FUNCTION_BLOCK PUBLIC TOD_TO_TestSuite EXTENDS TcUnit.FB_TestSuite
VAR
END_VAR

Check_TOD_TO_BOOL_Max();
Check_TOD_TO_BOOL_Min();
Check_TOD_TO_BYTE_Max();
Check_TOD_TO_BYTE_Min();
Check_TOD_TO_BYTE_TooHigh();
Check_TOD_TO_WORD_Max();
Check_TOD_TO_WORD_Min();
Check_TOD_TO_WORD_TooHigh();
Check_TOD_TO_DWORD_Max();
Check_TOD_TO_DWORD_Min();
Check_TOD_TO_LWORD_Max();
Check_TOD_TO_LWORD_Min();
Check_TOD_TO_SINT_Max();
Check_TOD_TO_SINT_Min();
Check_TOD_TO_SINT_TooHigh();
Check_TOD_TO_INT_Max();
Check_TOD_TO_INT_Min();
Check_TOD_TO_INT_TooHigh();
Check_TOD_TO_DINT_Max();
Check_TOD_TO_DINT_Min();
Check_TOD_TO_LINT_Max();
Check_TOD_TO_LINT_Min();
Check_TOD_TO_USINT_Max();
Check_TOD_TO_USINT_Min();
Check_TOD_TO_USINT_TooHigh();
Check_TOD_TO_UINT_Max();
Check_TOD_TO_UINT_Min();
Check_TOD_TO_UINT_TooHigh();
Check_TOD_TO_UDINT_Max();
Check_TOD_TO_UDINT_Min();
Check_TOD_TO_ULINT_Max();
Check_TOD_TO_ULINT_Min();
Check_TOD_TO_REAL_Max();
Check_TOD_TO_REAL_Min();
Check_TOD_TO_LREAL_Max();
Check_TOD_TO_LREAL_Min();
Check_TOD_TO_TIME_Max();
Check_TOD_TO_TIME_Min();
Check_TOD_TO_TOD_Max();
Check_TOD_TO_TOD_Min();
Check_TOD_TO_DATE_Max();
Check_TOD_TO_DATE_Min();
Check_TOD_TO_DT_Max();
Check_TOD_TO_DT_Min();
Check_TOD_TO_STRING_Max();
Check_TOD_TO_STRING_Min();

METHOD PUBLIC Check_TOD_TO_BOOL_Min
VAR
	value : TOD := DatatypeLimits.TOD_MIN_VALUE;
	actual : BOOL;
	converted : BOOL;
	equal : BOOL;
END_VAR
TEST('Check_TOD_TO_BOOL_Min');

// @TEST-RUN
converted := TryConvert_TOD_TO_Destination(value, actual);
equal := actual = TOD_TO_BOOL(value);

// @TEST-ASSERT
AssertTrue(Condition := equal, Message := 'Did not convert TOD to BOOL correctly');
AssertTrue(Condition := converted, Message := 'Did not report TOD to BOOL conversion was successful');

TEST_FINISHED();
END_METHOD

METHOD PUBLIC Check_TOD_TO_BOOL_Max
VAR
	value : TOD := DatatypeLimits.TOD_MAX_VALUE;
	actual : BOOL;
	converted : BOOL;
	equal : BOOL;
END_VAR
TEST('Check_TOD_TO_BOOL_Max');

// @TEST-RUN
converted := TryConvert_TOD_TO_Destination(value, actual);
equal := actual = TOD_TO_BOOL(value);

// @TEST-ASSERT
AssertTrue(Condition := equal, Message := 'Did not convert TOD to BOOL correctly');
AssertTrue(Condition := converted, Message := 'Did not report TOD to BOOL conversion was successful');

TEST_FINISHED();
END_METHOD

METHOD PUBLIC Check_TOD_TO_BYTE_Min
VAR
	value : TOD := DatatypeLimits.TOD_MIN_VALUE;
	actual : BYTE;
	converted : BOOL;
	equal : BOOL;
END_VAR
TEST('Check_TOD_TO_BYTE_Min');

// @TEST-RUN
converted := TryConvert_TOD_TO_Destination(value, actual);
equal := actual = TOD_TO_BYTE(value);

// @TEST-ASSERT
AssertTrue(Condition := equal, Message := 'Did not convert TOD to BYTE correctly');
AssertTrue(Condition := converted, Message := 'Did not report TOD to BYTE conversion was successful');

TEST_FINISHED();
END_METHOD

METHOD PUBLIC Check_TOD_TO_BYTE_TooHigh
VAR
	value : TOD := DatatypeLimits.TOD_MAX_VALUE;
	actual : BYTE;
	converted : BOOL;
END_VAR
TEST('Check_TOD_TO_BYTE_TooHigh');

// @TEST-RUN
converted := TryConvert_TOD_TO_Destination(value, actual);

// @TEST-ASSERT
AssertFalse(Condition := converted, Message := 'Did not report TOD to BYTE conversion was prevented');

TEST_FINISHED();
END_METHOD

METHOD PUBLIC Check_TOD_TO_BYTE_Max
VAR
	value : TOD := DatatypeLimits.MAX_VALUE_OF_TOD_WHICH_CAN_BE_HELD_IN_A_BYTE;
	actual : BYTE;
	converted : BOOL;
	equal : BOOL;
END_VAR
TEST('Check_TOD_TO_BYTE_Max');

// @TEST-RUN
converted := TryConvert_TOD_TO_Destination(value, actual);
equal := actual = TOD_TO_BYTE(value);

// @TEST-ASSERT
AssertTrue(Condition := equal, Message := 'Did not convert TOD to BYTE correctly');
AssertTrue(Condition := converted, Message := 'Did not report TOD to BYTE conversion was successful');

TEST_FINISHED();
END_METHOD

METHOD PUBLIC Check_TOD_TO_DATE_Min
VAR
	value : TOD := DatatypeLimits.TOD_MIN_VALUE;
	actual : DATE;
	converted : BOOL;
	equal : BOOL;
END_VAR
TEST('Check_TOD_TO_DATE_Min');

// @TEST-RUN
converted := TryConvert_TOD_TO_Destination(value, actual);
equal := actual = TOD_TO_DATE(value);

// @TEST-ASSERT
AssertTrue(Condition := equal, Message := 'Did not convert TOD to DATE correctly');
AssertTrue(Condition := converted, Message := 'Did not report TOD to DATE conversion was successful');

TEST_FINISHED();
END_METHOD

METHOD PUBLIC Check_TOD_TO_DATE_Max
VAR
	value : TOD := DatatypeLimits.TOD_MAX_VALUE;
	actual : DATE;
	converted : BOOL;
	equal : BOOL;
END_VAR
TEST('Check_TOD_TO_DATE_Max');

// @TEST-RUN
converted := TryConvert_TOD_TO_Destination(value, actual);
equal := actual = TOD_TO_DATE(value);

// @TEST-ASSERT
AssertTrue(Condition := equal, Message := 'Did not convert TOD to DATE correctly');
AssertTrue(Condition := converted, Message := 'Did not report TOD to DATE conversion was successful');

TEST_FINISHED();
END_METHOD

METHOD PUBLIC Check_TOD_TO_DINT_Min
VAR
	value : TOD := DatatypeLimits.TOD_MIN_VALUE;
	actual : DINT;
	converted : BOOL;
	equal : BOOL;
END_VAR
TEST('Check_TOD_TO_DINT_Min');

// @TEST-RUN
converted := TryConvert_TOD_TO_Destination(value, actual);
equal := actual = TOD_TO_DINT(value);

// @TEST-ASSERT
AssertTrue(Condition := equal, Message := 'Did not convert TOD to DINT correctly');
AssertTrue(Condition := converted, Message := 'Did not report TOD to DINT conversion was successful');

TEST_FINISHED();
END_METHOD

METHOD PUBLIC Check_TOD_TO_DINT_Max
VAR
	value : TOD := DatatypeLimits.TOD_MAX_VALUE;
	actual : DINT;
	converted : BOOL;
	equal : BOOL;
END_VAR
TEST('Check_TOD_TO_DINT_Max');

// @TEST-RUN
converted := TryConvert_TOD_TO_Destination(value, actual);
equal := actual = TOD_TO_DINT(value);

// @TEST-ASSERT
AssertTrue(Condition := equal, Message := 'Did not convert TOD to DINT correctly');
AssertTrue(Condition := converted, Message := 'Did not report TOD to DINT conversion was successful');

TEST_FINISHED();
END_METHOD

METHOD PUBLIC Check_TOD_TO_DT_Min
VAR
	value : TOD := DatatypeLimits.TOD_MIN_VALUE;
	actual : DT;
	converted : BOOL;
	equal : BOOL;
END_VAR
TEST('Check_TOD_TO_DT_Min');

// @TEST-RUN
converted := TryConvert_TOD_TO_Destination(value, actual);
equal := actual = TOD_TO_DT(value);

// @TEST-ASSERT
AssertTrue(Condition := equal, Message := 'Did not convert TOD to DT correctly');
AssertTrue(Condition := converted, Message := 'Did not report TOD to DT conversion was successful');

TEST_FINISHED();
END_METHOD

METHOD PUBLIC Check_TOD_TO_DT_Max
VAR
	value : TOD := DatatypeLimits.TOD_MAX_VALUE;
	actual : DT;
	converted : BOOL;
	equal : BOOL;
END_VAR
TEST('Check_TOD_TO_DT_Max');

// @TEST-RUN
converted := TryConvert_TOD_TO_Destination(value, actual);
equal := actual = TOD_TO_DT(value);

// @TEST-ASSERT
AssertTrue(Condition := equal, Message := 'Did not convert TOD to DT correctly');
AssertTrue(Condition := converted, Message := 'Did not report TOD to DT conversion was successful');

TEST_FINISHED();
END_METHOD

METHOD PUBLIC Check_TOD_TO_DWORD_Min
VAR
	value : TOD := DatatypeLimits.TOD_MIN_VALUE;
	actual : DWORD;
	converted : BOOL;
	equal : BOOL;
END_VAR
TEST('Check_TOD_TO_DWORD_Min');

// @TEST-RUN
converted := TryConvert_TOD_TO_Destination(value, actual);
equal := actual = TOD_TO_DWORD(value);

// @TEST-ASSERT
AssertTrue(Condition := equal, Message := 'Did not convert TOD to DWORD correctly');
AssertTrue(Condition := converted, Message := 'Did not report TOD to DWORD conversion was successful');

TEST_FINISHED();
END_METHOD

METHOD PUBLIC Check_TOD_TO_DWORD_Max
VAR
	value : TOD := DatatypeLimits.TOD_MAX_VALUE;
	actual : DWORD;
	converted : BOOL;
	equal : BOOL;
END_VAR
TEST('Check_TOD_TO_DWORD_Max');

// @TEST-RUN
converted := TryConvert_TOD_TO_Destination(value, actual);
equal := actual = TOD_TO_DWORD(value);

// @TEST-ASSERT
AssertTrue(Condition := equal, Message := 'Did not convert TOD to DWORD correctly');
AssertTrue(Condition := converted, Message := 'Did not report TOD to DWORD conversion was successful');

TEST_FINISHED();
END_METHOD

METHOD PUBLIC Check_TOD_TO_INT_Min
VAR
	value : TOD := DatatypeLimits.TOD_MIN_VALUE;
	actual : INT;
	converted : BOOL;
	equal : BOOL;
END_VAR
TEST('Check_TOD_TO_INT_Min');

// @TEST-RUN
converted := TryConvert_TOD_TO_Destination(value, actual);
equal := actual = TOD_TO_INT(value);

// @TEST-ASSERT
AssertTrue(Condition := equal, Message := 'Did not convert TOD to INT correctly');
AssertTrue(Condition := converted, Message := 'Did not report TOD to INT conversion was successful');

TEST_FINISHED();
END_METHOD

METHOD PUBLIC Check_TOD_TO_INT_TooHigh
VAR
	value : TOD := DatatypeLimits.TOD_MAX_VALUE;
	actual : INT;
	converted : BOOL;
END_VAR
TEST('Check_TOD_TO_INT_TooHigh');

// @TEST-RUN
converted := TryConvert_TOD_TO_Destination(value, actual);

// @TEST-ASSERT
AssertFalse(Condition := converted, Message := 'Did not report TOD to INT conversion was prevented');

TEST_FINISHED();
END_METHOD

METHOD PUBLIC Check_TOD_TO_INT_Max
VAR
	value : TOD := DatatypeLimits.MAX_VALUE_OF_TOD_WHICH_CAN_BE_HELD_IN_A_INT;
	actual : INT;
	converted : BOOL;
	equal : BOOL;
END_VAR
TEST('Check_TOD_TO_INT_Max');

// @TEST-RUN
converted := TryConvert_TOD_TO_Destination(value, actual);
equal := actual = TOD_TO_INT(value);

// @TEST-ASSERT
AssertTrue(Condition := equal, Message := 'Did not convert TOD to INT correctly');
AssertTrue(Condition := converted, Message := 'Did not report TOD to INT conversion was successful');

TEST_FINISHED();
END_METHOD

METHOD PUBLIC Check_TOD_TO_LINT_Min
VAR
	value : TOD := DatatypeLimits.TOD_MIN_VALUE;
	actual : LINT;
	converted : BOOL;
	equal : BOOL;
END_VAR
TEST('Check_TOD_TO_LINT_Min');

// @TEST-RUN
converted := TryConvert_TOD_TO_Destination(value, actual);
equal := actual = TOD_TO_LINT(value);

// @TEST-ASSERT
AssertTrue(Condition := equal, Message := 'Did not convert TOD to LINT correctly');
AssertTrue(Condition := converted, Message := 'Did not report TOD to LINT conversion was successful');

TEST_FINISHED();
END_METHOD

METHOD PUBLIC Check_TOD_TO_LINT_Max
VAR
	value : TOD := DatatypeLimits.TOD_MAX_VALUE;
	actual : LINT;
	converted : BOOL;
	equal : BOOL;
END_VAR
TEST('Check_TOD_TO_LINT_Max');

// @TEST-RUN
converted := TryConvert_TOD_TO_Destination(value, actual);
equal := actual = TOD_TO_LINT(value);

// @TEST-ASSERT
AssertTrue(Condition := equal, Message := 'Did not convert TOD to LINT correctly');
AssertTrue(Condition := converted, Message := 'Did not report TOD to LINT conversion was successful');

TEST_FINISHED();
END_METHOD

METHOD PUBLIC Check_TOD_TO_LREAL_Min
VAR
	value : TOD := DatatypeLimits.TOD_MIN_VALUE;
	actual : LREAL;
	converted : BOOL;
	equal : BOOL;
END_VAR
TEST('Check_TOD_TO_LREAL_Min');

// @TEST-RUN
converted := TryConvert_TOD_TO_Destination(value, actual);
equal := actual = TOD_TO_LREAL(value);

// @TEST-ASSERT
AssertTrue(Condition := equal, Message := 'Did not convert TOD to LREAL correctly');
AssertTrue(Condition := converted, Message := 'Did not report TOD to LREAL conversion was successful');

TEST_FINISHED();
END_METHOD

METHOD PUBLIC Check_TOD_TO_LREAL_Max
VAR
	value : TOD := DatatypeLimits.TOD_MAX_VALUE;
	actual : LREAL;
	converted : BOOL;
	equal : BOOL;
END_VAR
TEST('Check_TOD_TO_LREAL_Max');

// @TEST-RUN
converted := TryConvert_TOD_TO_Destination(value, actual);
equal := actual = TOD_TO_LREAL(value);

// @TEST-ASSERT
AssertTrue(Condition := equal, Message := 'Did not convert TOD to LREAL correctly');
AssertTrue(Condition := converted, Message := 'Did not report TOD to LREAL conversion was successful');

TEST_FINISHED();
END_METHOD

METHOD PUBLIC Check_TOD_TO_LWORD_Min
VAR
	value : TOD := DatatypeLimits.TOD_MIN_VALUE;
	actual : LWORD;
	converted : BOOL;
	equal : BOOL;
END_VAR
TEST('Check_TOD_TO_LWORD_Min');

// @TEST-RUN
converted := TryConvert_TOD_TO_Destination(value, actual);
equal := actual = TOD_TO_LWORD(value);

// @TEST-ASSERT
AssertTrue(Condition := equal, Message := 'Did not convert TOD to LWORD correctly');
AssertTrue(Condition := converted, Message := 'Did not report TOD to LWORD conversion was successful');

TEST_FINISHED();
END_METHOD

METHOD PUBLIC Check_TOD_TO_LWORD_Max
VAR
	value : TOD := DatatypeLimits.TOD_MAX_VALUE;
	actual : LWORD;
	converted : BOOL;
	equal : BOOL;
END_VAR
TEST('Check_TOD_TO_LWORD_Max');

// @TEST-RUN
converted := TryConvert_TOD_TO_Destination(value, actual);
equal := actual = TOD_TO_LWORD(value);

// @TEST-ASSERT
AssertTrue(Condition := equal, Message := 'Did not convert TOD to LWORD correctly');
AssertTrue(Condition := converted, Message := 'Did not report TOD to LWORD conversion was successful');

TEST_FINISHED();
END_METHOD

METHOD PUBLIC Check_TOD_TO_REAL_Min
VAR
	value : TOD := DatatypeLimits.TOD_MIN_VALUE;
	actual : REAL;
	converted : BOOL;
	equal : BOOL;
END_VAR
TEST('Check_TOD_TO_REAL_Min');

// @TEST-RUN
converted := TryConvert_TOD_TO_Destination(value, actual);
equal := actual = TOD_TO_REAL(value);

// @TEST-ASSERT
AssertTrue(Condition := equal, Message := 'Did not convert TOD to REAL correctly');
AssertTrue(Condition := converted, Message := 'Did not report TOD to REAL conversion was successful');

TEST_FINISHED();
END_METHOD

METHOD PUBLIC Check_TOD_TO_REAL_Max
VAR
	value : TOD := DatatypeLimits.TOD_MAX_VALUE;
	actual : REAL;
	converted : BOOL;
	equal : BOOL;
END_VAR
TEST('Check_TOD_TO_REAL_Max');

// @TEST-RUN
converted := TryConvert_TOD_TO_Destination(value, actual);
equal := actual = TOD_TO_REAL(value);

// @TEST-ASSERT
AssertTrue(Condition := equal, Message := 'Did not convert TOD to REAL correctly');
AssertTrue(Condition := converted, Message := 'Did not report TOD to REAL conversion was successful');

TEST_FINISHED();
END_METHOD

METHOD PUBLIC Check_TOD_TO_SINT_Min
VAR
	value : TOD := DatatypeLimits.TOD_MIN_VALUE;
	actual : SINT;
	converted : BOOL;
	equal : BOOL;
END_VAR
TEST('Check_TOD_TO_SINT_Min');

// @TEST-RUN
converted := TryConvert_TOD_TO_Destination(value, actual);
equal := actual = TOD_TO_SINT(value);

// @TEST-ASSERT
AssertTrue(Condition := equal, Message := 'Did not convert TOD to SINT correctly');
AssertTrue(Condition := converted, Message := 'Did not report TOD to SINT conversion was successful');

TEST_FINISHED();
END_METHOD

METHOD PUBLIC Check_TOD_TO_SINT_TooHigh
VAR
	value : TOD := DatatypeLimits.TOD_MAX_VALUE;
	actual : SINT;
	converted : BOOL;
END_VAR
TEST('Check_TOD_TO_SINT_TooHigh');

// @TEST-RUN
converted := TryConvert_TOD_TO_Destination(value, actual);

// @TEST-ASSERT
AssertFalse(Condition := converted, Message := 'Did not report TOD to SINT conversion was prevented');

TEST_FINISHED();
END_METHOD

METHOD PUBLIC Check_TOD_TO_SINT_Max
VAR
	value : TOD := DatatypeLimits.MAX_VALUE_OF_TOD_WHICH_CAN_BE_HELD_IN_A_SINT;
	actual : SINT;
	converted : BOOL;
	equal : BOOL;
END_VAR
TEST('Check_TOD_TO_SINT_Max');

// @TEST-RUN
converted := TryConvert_TOD_TO_Destination(value, actual);
equal := actual = TOD_TO_SINT(value);

// @TEST-ASSERT
AssertTrue(Condition := equal, Message := 'Did not convert TOD to SINT correctly');
AssertTrue(Condition := converted, Message := 'Did not report TOD to SINT conversion was successful');

TEST_FINISHED();
END_METHOD

METHOD PUBLIC Check_TOD_TO_STRING_Min
VAR
	value : TOD := DatatypeLimits.TOD_MIN_VALUE;
	actual : STRING;
	converted : BOOL;
	equal : BOOL;
END_VAR
TEST('Check_TOD_TO_STRING_Min');

// @TEST-RUN
converted := TryConvert_TOD_TO_Destination(value, actual);
equal := actual = TOD_TO_STRING(value);

// @TEST-ASSERT
AssertTrue(Condition := equal, Message := 'Did not convert TOD to STRING correctly');
AssertTrue(Condition := converted, Message := 'Did not report TOD to STRING conversion was successful');

TEST_FINISHED();
END_METHOD

METHOD PUBLIC Check_TOD_TO_STRING_Max
VAR
	value : TOD := DatatypeLimits.TOD_MAX_VALUE;
	actual : STRING;
	converted : BOOL;
	equal : BOOL;
END_VAR
TEST('Check_TOD_TO_STRING_Max');

// @TEST-RUN
converted := TryConvert_TOD_TO_Destination(value, actual);
equal := actual = TOD_TO_STRING(value);

// @TEST-ASSERT
AssertTrue(Condition := equal, Message := 'Did not convert TOD to STRING correctly');
AssertTrue(Condition := converted, Message := 'Did not report TOD to STRING conversion was successful');

TEST_FINISHED();
END_METHOD

METHOD PUBLIC Check_TOD_TO_TIME_Min
VAR
	value : TOD := DatatypeLimits.TOD_MIN_VALUE;
	actual : TIME;
	converted : BOOL;
	equal : BOOL;
END_VAR
TEST('Check_TOD_TO_TIME_Min');

// @TEST-RUN
converted := TryConvert_TOD_TO_Destination(value, actual);
equal := actual = TOD_TO_TIME(value);

// @TEST-ASSERT
AssertTrue(Condition := equal, Message := 'Did not convert TOD to TIME correctly');
AssertTrue(Condition := converted, Message := 'Did not report TOD to TIME conversion was successful');

TEST_FINISHED();
END_METHOD

METHOD PUBLIC Check_TOD_TO_TIME_Max
VAR
	value : TOD := DatatypeLimits.TOD_MAX_VALUE;
	actual : TIME;
	converted : BOOL;
	equal : BOOL;
END_VAR
TEST('Check_TOD_TO_TIME_Max');

// @TEST-RUN
converted := TryConvert_TOD_TO_Destination(value, actual);
equal := actual = TOD_TO_TIME(value);

// @TEST-ASSERT
AssertTrue(Condition := equal, Message := 'Did not convert TOD to TIME correctly');
AssertTrue(Condition := converted, Message := 'Did not report TOD to TIME conversion was successful');

TEST_FINISHED();
END_METHOD

METHOD PUBLIC Check_TOD_TO_TOD_Min
VAR
	value : TOD := DatatypeLimits.TOD_MIN_VALUE;
	actual : TOD;
	converted : BOOL;
	equal : BOOL;
END_VAR
TEST('Check_TOD_TO_TOD_Min');

// @TEST-RUN
converted := TryConvert_TOD_TO_Destination(value, actual);
equal := actual = value;

// @TEST-ASSERT
AssertTrue(Condition := equal, Message := 'Did not convert TOD to TOD correctly');
AssertTrue(Condition := converted, Message := 'Did not report TOD to TOD conversion was successful');

TEST_FINISHED();
END_METHOD

METHOD PUBLIC Check_TOD_TO_TOD_Max
VAR
	value : TOD := DatatypeLimits.TOD_MAX_VALUE;
	actual : TOD;
	converted : BOOL;
	equal : BOOL;
END_VAR
TEST('Check_TOD_TO_TOD_Max');

// @TEST-RUN
converted := TryConvert_TOD_TO_Destination(value, actual);
equal := actual = value;

// @TEST-ASSERT
AssertTrue(Condition := equal, Message := 'Did not convert TOD to TOD correctly');
AssertTrue(Condition := converted, Message := 'Did not report TOD to TOD conversion was successful');

TEST_FINISHED();
END_METHOD

METHOD PUBLIC Check_TOD_TO_UDINT_Min
VAR
	value : TOD := DatatypeLimits.TOD_MIN_VALUE;
	actual : UDINT;
	converted : BOOL;
	equal : BOOL;
END_VAR
TEST('Check_TOD_TO_UDINT_Min');

// @TEST-RUN
converted := TryConvert_TOD_TO_Destination(value, actual);
equal := actual = TOD_TO_UDINT(value);

// @TEST-ASSERT
AssertTrue(Condition := equal, Message := 'Did not convert TOD to UDINT correctly');
AssertTrue(Condition := converted, Message := 'Did not report TOD to UDINT conversion was successful');

TEST_FINISHED();
END_METHOD

METHOD PUBLIC Check_TOD_TO_UDINT_Max
VAR
	value : TOD := DatatypeLimits.TOD_MAX_VALUE;
	actual : UDINT;
	converted : BOOL;
	equal : BOOL;
END_VAR
TEST('Check_TOD_TO_UDINT_Max');

// @TEST-RUN
converted := TryConvert_TOD_TO_Destination(value, actual);
equal := actual = TOD_TO_UDINT(value);

// @TEST-ASSERT
AssertTrue(Condition := equal, Message := 'Did not convert TOD to UDINT correctly');
AssertTrue(Condition := converted, Message := 'Did not report TOD to UDINT conversion was successful');

TEST_FINISHED();
END_METHOD

METHOD PUBLIC Check_TOD_TO_UINT_Min
VAR
	value : TOD := DatatypeLimits.TOD_MIN_VALUE;
	actual : UINT;
	converted : BOOL;
	equal : BOOL;
END_VAR
TEST('Check_TOD_TO_UINT_Min');

// @TEST-RUN
converted := TryConvert_TOD_TO_Destination(value, actual);
equal := actual = TOD_TO_UINT(value);

// @TEST-ASSERT
AssertTrue(Condition := equal, Message := 'Did not convert TOD to UINT correctly');
AssertTrue(Condition := converted, Message := 'Did not report TOD to UINT conversion was successful');

TEST_FINISHED();
END_METHOD

METHOD PUBLIC Check_TOD_TO_UINT_TooHigh
VAR
	value : TOD := DatatypeLimits.TOD_MAX_VALUE;
	actual : UINT;
	converted : BOOL;
END_VAR
TEST('Check_TOD_TO_UINT_TooHigh');

// @TEST-RUN
converted := TryConvert_TOD_TO_Destination(value, actual);

// @TEST-ASSERT
AssertFalse(Condition := converted, Message := 'Did not report TOD to UINT conversion was prevented');

TEST_FINISHED();
END_METHOD

METHOD PUBLIC Check_TOD_TO_UINT_Max
VAR
	value : TOD := DatatypeLimits.MAX_VALUE_OF_TOD_WHICH_CAN_BE_HELD_IN_A_UINT;
	actual : UINT;
	converted : BOOL;
	equal : BOOL;
END_VAR
TEST('Check_TOD_TO_UINT_Max');

// @TEST-RUN
converted := TryConvert_TOD_TO_Destination(value, actual);
equal := actual = TOD_TO_UINT(value);

// @TEST-ASSERT
AssertTrue(Condition := equal, Message := 'Did not convert TOD to UINT correctly');
AssertTrue(Condition := converted, Message := 'Did not report TOD to UINT conversion was successful');

TEST_FINISHED();
END_METHOD

METHOD PUBLIC Check_TOD_TO_ULINT_Min
VAR
	value : TOD := DatatypeLimits.TOD_MIN_VALUE;
	actual : ULINT;
	converted : BOOL;
	equal : BOOL;
END_VAR
TEST('Check_TOD_TO_ULINT_Min');

// @TEST-RUN
converted := TryConvert_TOD_TO_Destination(value, actual);
equal := actual = TOD_TO_ULINT(value);

// @TEST-ASSERT
AssertTrue(Condition := equal, Message := 'Did not convert TOD to ULINT correctly');
AssertTrue(Condition := converted, Message := 'Did not report TOD to ULINT conversion was successful');

TEST_FINISHED();
END_METHOD

METHOD PUBLIC Check_TOD_TO_ULINT_Max
VAR
	value : TOD := DatatypeLimits.TOD_MAX_VALUE;
	actual : ULINT;
	converted : BOOL;
	equal : BOOL;
END_VAR
TEST('Check_TOD_TO_ULINT_Max');

// @TEST-RUN
converted := TryConvert_TOD_TO_Destination(value, actual);
equal := actual = TOD_TO_ULINT(value);

// @TEST-ASSERT
AssertTrue(Condition := equal, Message := 'Did not convert TOD to ULINT correctly');
AssertTrue(Condition := converted, Message := 'Did not report TOD to ULINT conversion was successful');

TEST_FINISHED();
END_METHOD

METHOD PUBLIC Check_TOD_TO_USINT_Min
VAR
	value : TOD := DatatypeLimits.TOD_MIN_VALUE;
	actual : USINT;
	converted : BOOL;
	equal : BOOL;
END_VAR
TEST('Check_TOD_TO_USINT_Min');

// @TEST-RUN
converted := TryConvert_TOD_TO_Destination(value, actual);
equal := actual = TOD_TO_USINT(value);

// @TEST-ASSERT
AssertTrue(Condition := equal, Message := 'Did not convert TOD to USINT correctly');
AssertTrue(Condition := converted, Message := 'Did not report TOD to USINT conversion was successful');

TEST_FINISHED();
END_METHOD

METHOD PUBLIC Check_TOD_TO_USINT_TooHigh
VAR
	value : TOD := DatatypeLimits.TOD_MAX_VALUE;
	actual : USINT;
	converted : BOOL;
END_VAR
TEST('Check_TOD_TO_USINT_TooHigh');

// @TEST-RUN
converted := TryConvert_TOD_TO_Destination(value, actual);

// @TEST-ASSERT
AssertFalse(Condition := converted, Message := 'Did not report TOD to USINT conversion was prevented');

TEST_FINISHED();
END_METHOD

METHOD PUBLIC Check_TOD_TO_USINT_Max
VAR
	value : TOD := DatatypeLimits.MAX_VALUE_OF_TOD_WHICH_CAN_BE_HELD_IN_A_USINT;
	actual : USINT;
	converted : BOOL;
	equal : BOOL;
END_VAR
TEST('Check_TOD_TO_USINT_Max');

// @TEST-RUN
converted := TryConvert_TOD_TO_Destination(value, actual);
equal := actual = TOD_TO_USINT(value);

// @TEST-ASSERT
AssertTrue(Condition := equal, Message := 'Did not convert TOD to USINT correctly');
AssertTrue(Condition := converted, Message := 'Did not report TOD to USINT conversion was successful');

TEST_FINISHED();
END_METHOD

METHOD PUBLIC Check_TOD_TO_WORD_Min
VAR
	value : TOD := DatatypeLimits.TOD_MIN_VALUE;
	actual : WORD;
	converted : BOOL;
	equal : BOOL;
END_VAR
TEST('Check_TOD_TO_WORD_Min');

// @TEST-RUN
converted := TryConvert_TOD_TO_Destination(value, actual);
equal := actual = TOD_TO_WORD(value);

// @TEST-ASSERT
AssertTrue(Condition := equal, Message := 'Did not convert TOD to WORD correctly');
AssertTrue(Condition := converted, Message := 'Did not report TOD to WORD conversion was successful');

TEST_FINISHED();
END_METHOD

METHOD PUBLIC Check_TOD_TO_WORD_TooHigh
VAR
	value : TOD := DatatypeLimits.TOD_MAX_VALUE;
	actual : WORD;
	converted : BOOL;
END_VAR
TEST('Check_TOD_TO_WORD_TooHigh');

// @TEST-RUN
converted := TryConvert_TOD_TO_Destination(value, actual);

// @TEST-ASSERT
AssertFalse(Condition := converted, Message := 'Did not report TOD to WORD conversion was prevented');

TEST_FINISHED();
END_METHOD

METHOD PUBLIC Check_TOD_TO_WORD_Max
VAR
	value : TOD := DatatypeLimits.MAX_VALUE_OF_TOD_WHICH_CAN_BE_HELD_IN_A_WORD;
	actual : WORD;
	converted : BOOL;
	equal : BOOL;
END_VAR
TEST('Check_TOD_TO_WORD_Max');

// @TEST-RUN
converted := TryConvert_TOD_TO_Destination(value, actual);
equal := actual = TOD_TO_WORD(value);

// @TEST-ASSERT
AssertTrue(Condition := equal, Message := 'Did not convert TOD to WORD correctly');
AssertTrue(Condition := converted, Message := 'Did not report TOD to WORD conversion was successful');

TEST_FINISHED();
END_METHOD

END_FUNCTION_BLOCK

(* stored: Version 1.1.0.1, ProductVersion 3.1.4024.12
   POU TOD_TO_TestSuite: Id {268fba33-c979-45d2-9197-3ae649925bde}, SpecialFunc None
   Method Check_TOD_TO_BOOL_Min: Id {aa227d84-f942-4487-8b06-d71c2117467e}
   Method Check_TOD_TO_BOOL_Max: Id {ccc2f7bd-7b2e-43f1-8674-e826263e7839}
   Method Check_TOD_TO_BYTE_Min: Id {6f198f43-59b9-4a1b-93ba-d1f2f48c8840}
   Method Check_TOD_TO_BYTE_TooHigh: Id {9a1f85d9-5915-4371-8bd6-b4f15a804d4c}
   Method Check_TOD_TO_BYTE_Max: Id {cab93a36-8258-4b85-8e79-899116ff1600}
   Method Check_TOD_TO_DATE_Min: Id {567d70bc-6dd6-4538-83e5-06a6aabdd983}
   Method Check_TOD_TO_DATE_Max: Id {573ec20e-7917-46b7-9152-926daba2c265}
   Method Check_TOD_TO_DINT_Min: Id {58caaaf9-eb62-4db2-98eb-fa1d00ef2e06}
   Method Check_TOD_TO_DINT_Max: Id {b6c85a11-5adc-4f6f-9728-88152a5cae97}
   Method Check_TOD_TO_DT_Min: Id {13967396-aaa5-49b2-9268-7b41e800760a}
   Method Check_TOD_TO_DT_Max: Id {c316eea4-42f2-48ab-970b-fa0a5c6bc5ed}
   Method Check_TOD_TO_DWORD_Min: Id {0844839f-0f43-45ab-8ddd-028cc9b82f4d}
   Method Check_TOD_TO_DWORD_Max: Id {5c98d806-c971-4fc1-9516-7942a12181f3}
   Method Check_TOD_TO_INT_Min: Id {88bd3fbd-640f-4ba7-b434-32c1dcdb71ef}
   Method Check_TOD_TO_INT_TooHigh: Id {0e48184b-0607-436d-9932-b3a0e586c2a0}
   Method Check_TOD_TO_INT_Max: Id {6b3dd9b3-4ed5-4f0a-ad5a-e35767fe23b0}
   Method Check_TOD_TO_LINT_Min: Id {2992f989-dbec-4a8b-ad06-585f2aa69351}
   Method Check_TOD_TO_LINT_Max: Id {de08a0c7-eeb6-4b97-af35-882f9b0a7a7b}
   Method Check_TOD_TO_LREAL_Min: Id {1690aa2c-095f-4cd9-86a6-7923ff4e36f1}
   Method Check_TOD_TO_LREAL_Max: Id {3d5a8527-2a0a-4497-8264-4186364b4885}
   Method Check_TOD_TO_LWORD_Min: Id {fec9adc4-ae92-4dd4-830b-a6b007e3de55}
   Method Check_TOD_TO_LWORD_Max: Id {1714032a-9c16-4125-ae63-d1219e47d768}
   Method Check_TOD_TO_REAL_Min: Id {0624d10e-98c7-4864-879c-6921e623a8c4}
   Method Check_TOD_TO_REAL_Max: Id {23f57be8-1dff-40ae-8b3b-5466330f8bd1}
   Method Check_TOD_TO_SINT_Min: Id {429947b0-3dc6-4cee-8bdf-ad0b211331ce}
   Method Check_TOD_TO_SINT_TooHigh: Id {a3cc78ae-7c82-4ede-b25d-76fd567a9bc1}
   Method Check_TOD_TO_SINT_Max: Id {642d6359-89f4-40ef-8e11-bbf0cb63383d}
   Method Check_TOD_TO_STRING_Min: Id {a488fe9d-9e63-41b6-8219-8a5c0dfb2777}
   Method Check_TOD_TO_STRING_Max: Id {81b67ba5-3a7e-46d4-8069-78aba7d1e6cc}
   Method Check_TOD_TO_TIME_Min: Id {5ee7baaa-3c6f-4568-9a9e-630f198dff4d}
   Method Check_TOD_TO_TIME_Max: Id {134aef1e-1c88-439b-943f-785a2ed00b93}
   Method Check_TOD_TO_TOD_Min: Id {1ae14b25-3e55-40ef-a314-b54a5954d08c}
   Method Check_TOD_TO_TOD_Max: Id {c1ffd7b1-554c-495f-b876-91b420d26ad1}
   Method Check_TOD_TO_UDINT_Min: Id {2ad476d2-5821-4d50-a3ba-ce0e7c668d8c}
   Method Check_TOD_TO_UDINT_Max: Id {575fd89b-64cc-47e1-9891-6b4aef23af09}
   Method Check_TOD_TO_UINT_Min: Id {453d526d-b825-412f-8225-992e4e9be0d1}
   Method Check_TOD_TO_UINT_TooHigh: Id {163c68ae-9f1e-43f5-bb3f-87a9ceba03cf}
   Method Check_TOD_TO_UINT_Max: Id {88103e94-508b-4426-9a1c-58b66e8d2e79}
   Method Check_TOD_TO_ULINT_Min: Id {4d7d3ce1-4870-489f-9475-c5d2fa6d5d88}
   Method Check_TOD_TO_ULINT_Max: Id {04c2a8a5-5020-49fa-942f-86d058c4e9d4}
   Method Check_TOD_TO_USINT_Min: Id {f9e5db2f-44ec-469d-bc71-c7dd852fb350}
   Method Check_TOD_TO_USINT_TooHigh: Id {f0e20160-1b7e-45c5-b28e-b6a4c5f1813c}
   Method Check_TOD_TO_USINT_Max: Id {363eaa9f-958c-4d26-906a-a4a8382bb801}
   Method Check_TOD_TO_WORD_Min: Id {3a8bc1b0-a296-4008-9e5a-644679f63df6}
   Method Check_TOD_TO_WORD_TooHigh: Id {0d121ffa-9b55-4f05-ac96-eccae04f49c4}
   Method Check_TOD_TO_WORD_Max: Id {498a5923-b7f8-4fd1-9b9b-808e13723142} *)
